PROGRAM BLOCK_CALL
VAR
	CLAMP_1_DB : CLAMP_PROCESS;
	CLAMP_2_DB : CLAMP_PROCESS;
	CLAMP_3_DB : CLAMP_PROCESS;
	CLAMP_4_DB : CLAMP_PROCESS;
	CLAMP_5_DB : CLAMP_PROCESS;
	CLAMP_6_DB : CLAMP_PROCESS;
	Feedback_1_DB : Feedback_FB;
	Feedback_2_DB : Feedback_FB;
	Feedback_3_DB : Feedback_FB;
	Feedback_4_DB : Feedback_FB;
	Feedback_5_DB : Feedback_FB;
	Feedback_6_DB : Feedback_FB;
	Feedback_TT1_DB : Feedback_FB;
	Feedback_Trunion_1_DB : Feedback_FB;
	TURNTABLE_2POS_DB : TURNTABLE_2POS;
	TRUNION1_DB : TRUNION_FB;
	ROLLER_DOOR_DB : ROLLER_DOOR;
	RollerDoor_DB : RollerDoor;
    Feedback_RD1_DB : Feedback_FB;
	WELD_ROBOT_DB : WELD_ROBOT;
	MH_ROBOT_DB : MH_ROBOT;
	MODE_CONTROL_DB : MODE_CONTROL;
	SENSOR_DB : SENSOR;
END_VAR

// note: this text did not pass the execution check against the stored diagram
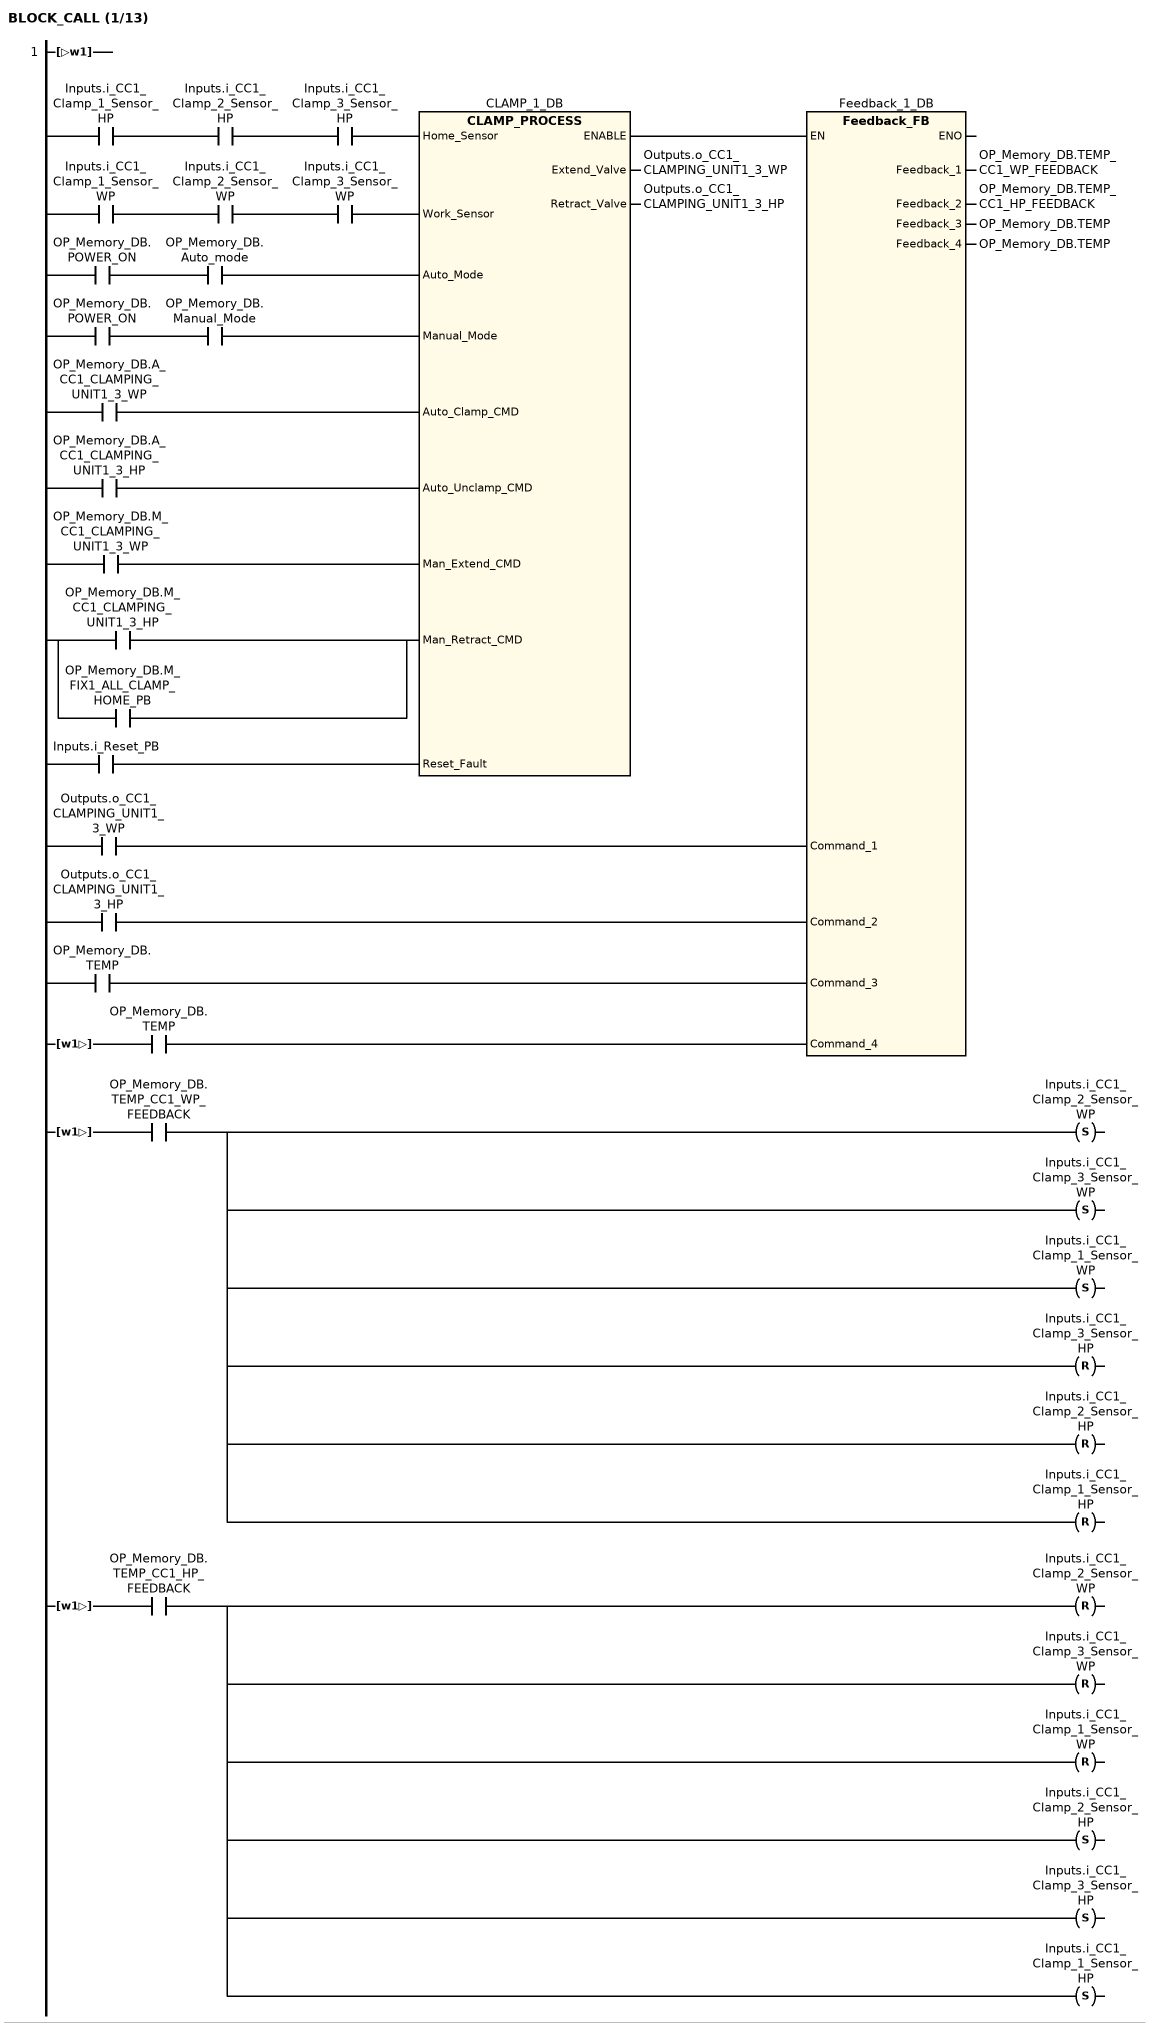
// NETWORK 1
CLAMP_1_DB(
    Home_Sensor := Inputs.i_CC1_Clamp_1_Sensor_HP AND Inputs.i_CC1_Clamp_2_Sensor_HP AND Inputs.i_CC1_Clamp_3_Sensor_HP,
    Work_Sensor := Inputs.i_CC1_Clamp_1_Sensor_WP AND Inputs.i_CC1_Clamp_2_Sensor_WP AND Inputs.i_CC1_Clamp_3_Sensor_WP,
    Auto_Mode := OP_Memory_DB.POWER_ON AND OP_Memory_DB.Auto_mode,
    Manual_Mode := OP_Memory_DB.POWER_ON AND OP_Memory_DB.Manual_Mode,
    Auto_Clamp_CMD := OP_Memory_DB.A_CC1_CLAMPING_UNIT1_3_WP,
    Auto_Unclamp_CMD := OP_Memory_DB.A_CC1_CLAMPING_UNIT1_3_HP,
    Man_Extend_CMD := OP_Memory_DB.M_CC1_CLAMPING_UNIT1_3_WP,
    Man_Retract_CMD := OP_Memory_DB.M_CC1_CLAMPING_UNIT1_3_HP OR OP_Memory_DB.M_FIX1_ALL_CLAMP_HOME_PB,
    Reset_Fault := Inputs.i_Reset_PB,
    Extend_Valve => Outputs.o_CC1_CLAMPING_UNIT1_3_WP,
    Retract_Valve => Outputs.o_CC1_CLAMPING_UNIT1_3_HP); // CLAMP_PROCESS
Feedback_1_DB(
    EN := CLAMP_1_DB.ENABLE,
    Command_1 := Outputs.o_CC1_CLAMPING_UNIT1_3_WP,
    Command_2 := Outputs.o_CC1_CLAMPING_UNIT1_3_HP,
    Command_3 := OP_Memory_DB.TEMP,
    Command_4 := OP_Memory_DB.TEMP,
    Feedback_1 => OP_Memory_DB.TEMP_CC1_WP_FEEDBACK,
    Feedback_2 => OP_Memory_DB.TEMP_CC1_HP_FEEDBACK,
    Feedback_3 => OP_Memory_DB.TEMP,
    Feedback_4 => OP_Memory_DB.TEMP); // Feedback_FB
Inputs.i_CC1_Clamp_2_Sensor_WP S= OP_Memory_DB.TEMP_CC1_WP_FEEDBACK;
Inputs.i_CC1_Clamp_3_Sensor_WP S= OP_Memory_DB.TEMP_CC1_WP_FEEDBACK;
Inputs.i_CC1_Clamp_1_Sensor_WP S= OP_Memory_DB.TEMP_CC1_WP_FEEDBACK;
Inputs.i_CC1_Clamp_3_Sensor_HP R= OP_Memory_DB.TEMP_CC1_WP_FEEDBACK;
Inputs.i_CC1_Clamp_2_Sensor_HP R= OP_Memory_DB.TEMP_CC1_WP_FEEDBACK;
Inputs.i_CC1_Clamp_1_Sensor_HP R= OP_Memory_DB.TEMP_CC1_WP_FEEDBACK;
Inputs.i_CC1_Clamp_2_Sensor_WP R= OP_Memory_DB.TEMP_CC1_HP_FEEDBACK;
Inputs.i_CC1_Clamp_3_Sensor_WP R= OP_Memory_DB.TEMP_CC1_HP_FEEDBACK;
Inputs.i_CC1_Clamp_1_Sensor_WP R= OP_Memory_DB.TEMP_CC1_HP_FEEDBACK;
Inputs.i_CC1_Clamp_2_Sensor_HP S= OP_Memory_DB.TEMP_CC1_HP_FEEDBACK;
Inputs.i_CC1_Clamp_3_Sensor_HP S= OP_Memory_DB.TEMP_CC1_HP_FEEDBACK;
Inputs.i_CC1_Clamp_1_Sensor_HP S= OP_Memory_DB.TEMP_CC1_HP_FEEDBACK;

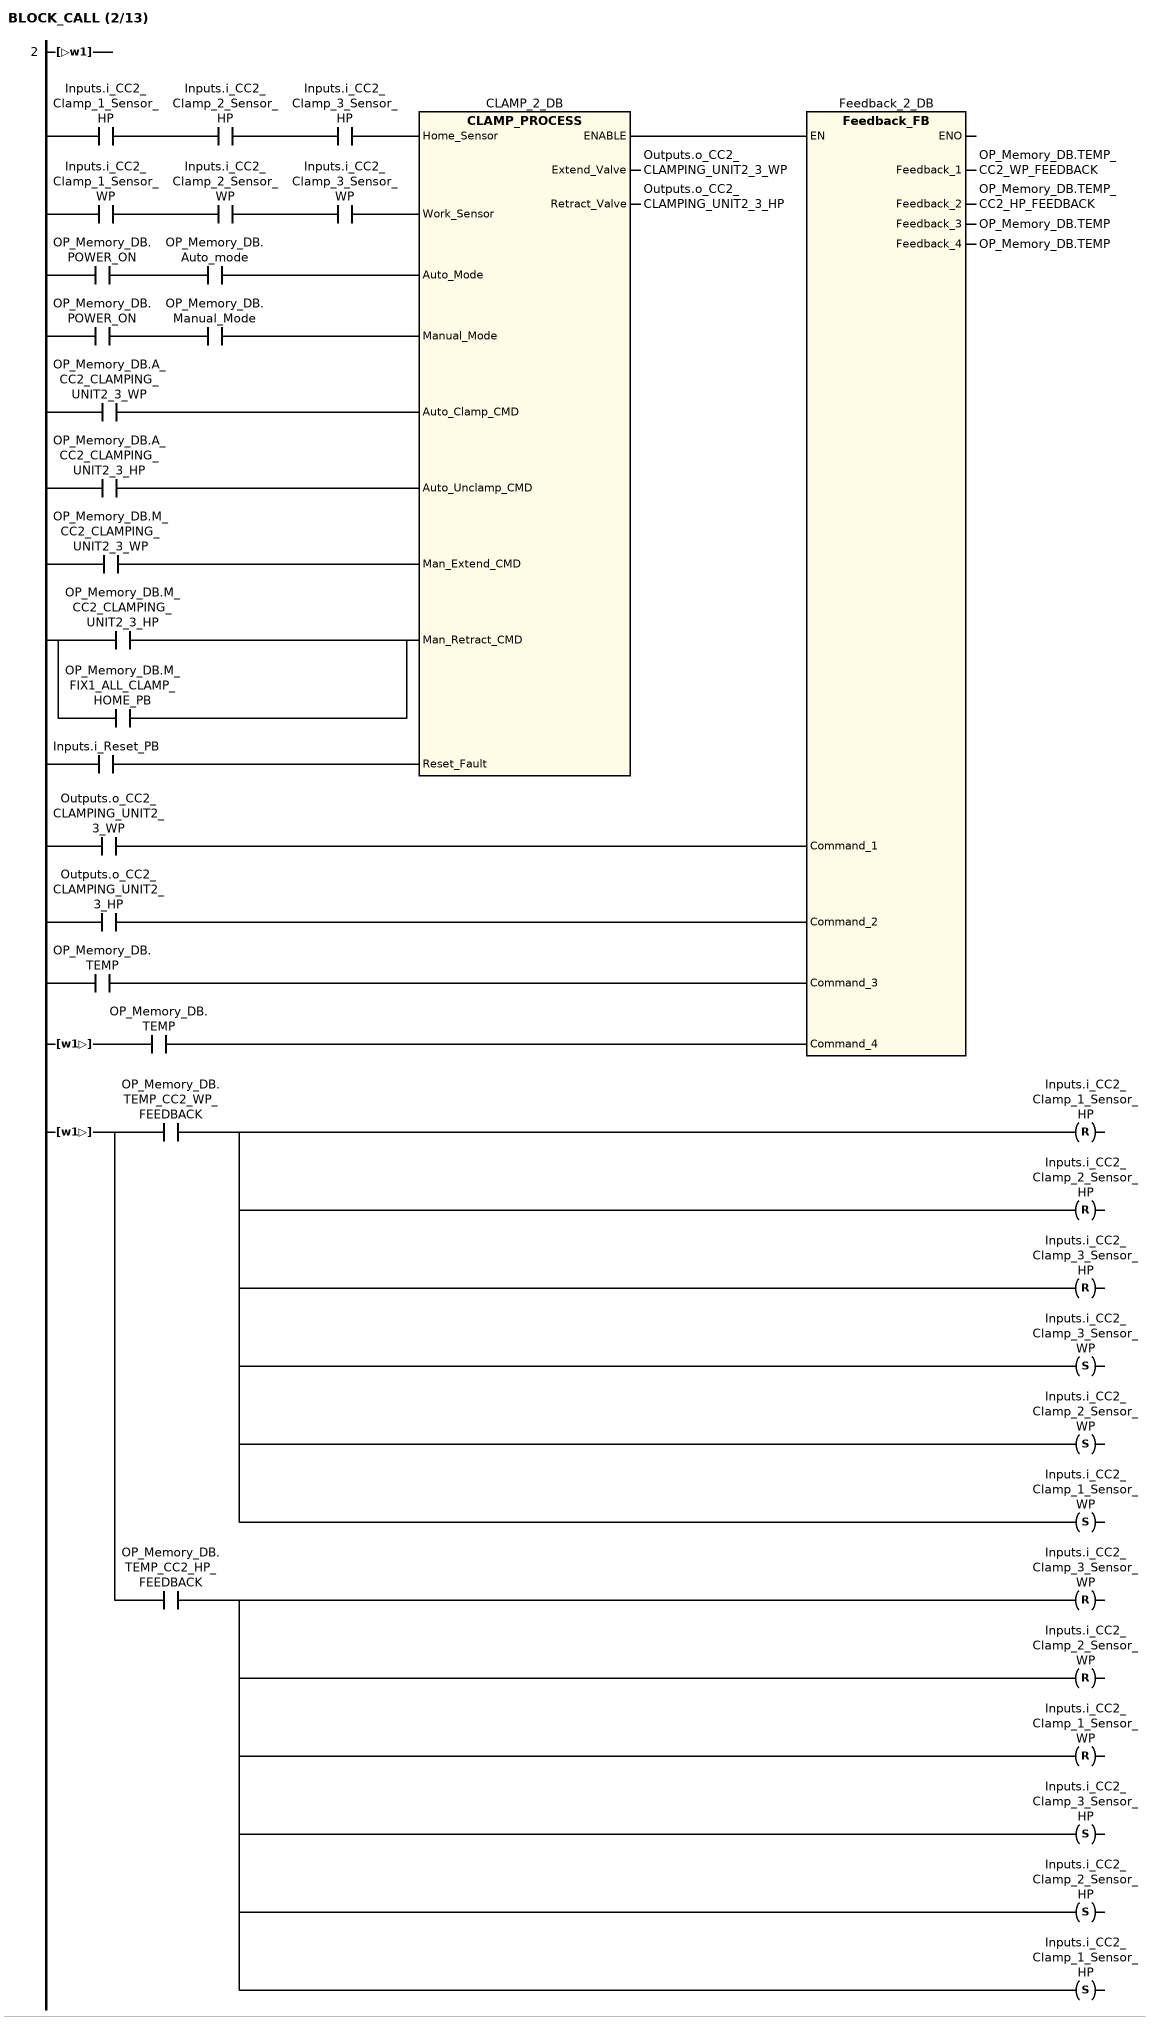
// NETWORK 2
CLAMP_2_DB(
    Home_Sensor := Inputs.i_CC2_Clamp_1_Sensor_HP AND Inputs.i_CC2_Clamp_2_Sensor_HP AND Inputs.i_CC2_Clamp_3_Sensor_HP,
    Work_Sensor := Inputs.i_CC2_Clamp_1_Sensor_WP AND Inputs.i_CC2_Clamp_2_Sensor_WP AND Inputs.i_CC2_Clamp_3_Sensor_WP,
    Auto_Mode := OP_Memory_DB.POWER_ON AND OP_Memory_DB.Auto_mode,
    Manual_Mode := OP_Memory_DB.POWER_ON AND OP_Memory_DB.Manual_Mode,
    Auto_Clamp_CMD := OP_Memory_DB.A_CC2_CLAMPING_UNIT2_3_WP,
    Auto_Unclamp_CMD := OP_Memory_DB.A_CC2_CLAMPING_UNIT2_3_HP,
    Man_Extend_CMD := OP_Memory_DB.M_CC2_CLAMPING_UNIT2_3_WP,
    Man_Retract_CMD := OP_Memory_DB.M_CC2_CLAMPING_UNIT2_3_HP OR OP_Memory_DB.M_FIX1_ALL_CLAMP_HOME_PB,
    Reset_Fault := Inputs.i_Reset_PB,
    Extend_Valve => Outputs.o_CC2_CLAMPING_UNIT2_3_WP,
    Retract_Valve => Outputs.o_CC2_CLAMPING_UNIT2_3_HP); // CLAMP_PROCESS
Feedback_2_DB(
    EN := CLAMP_2_DB.ENABLE,
    Command_1 := Outputs.o_CC2_CLAMPING_UNIT2_3_WP,
    Command_2 := Outputs.o_CC2_CLAMPING_UNIT2_3_HP,
    Command_3 := OP_Memory_DB.TEMP,
    Command_4 := OP_Memory_DB.TEMP,
    Feedback_1 => OP_Memory_DB.TEMP_CC2_WP_FEEDBACK,
    Feedback_2 => OP_Memory_DB.TEMP_CC2_HP_FEEDBACK,
    Feedback_3 => OP_Memory_DB.TEMP,
    Feedback_4 => OP_Memory_DB.TEMP); // Feedback_FB
Inputs.i_CC2_Clamp_1_Sensor_HP R= OP_Memory_DB.TEMP_CC2_WP_FEEDBACK;
Inputs.i_CC2_Clamp_2_Sensor_HP R= OP_Memory_DB.TEMP_CC2_WP_FEEDBACK;
Inputs.i_CC2_Clamp_3_Sensor_HP R= OP_Memory_DB.TEMP_CC2_WP_FEEDBACK;
Inputs.i_CC2_Clamp_3_Sensor_WP S= OP_Memory_DB.TEMP_CC2_WP_FEEDBACK;
Inputs.i_CC2_Clamp_2_Sensor_WP S= OP_Memory_DB.TEMP_CC2_WP_FEEDBACK;
Inputs.i_CC2_Clamp_1_Sensor_WP S= OP_Memory_DB.TEMP_CC2_WP_FEEDBACK;
Inputs.i_CC2_Clamp_3_Sensor_WP R= OP_Memory_DB.TEMP_CC2_HP_FEEDBACK;
Inputs.i_CC2_Clamp_2_Sensor_WP R= OP_Memory_DB.TEMP_CC2_HP_FEEDBACK;
Inputs.i_CC2_Clamp_1_Sensor_WP R= OP_Memory_DB.TEMP_CC2_HP_FEEDBACK;
Inputs.i_CC2_Clamp_3_Sensor_HP S= OP_Memory_DB.TEMP_CC2_HP_FEEDBACK;
Inputs.i_CC2_Clamp_2_Sensor_HP S= OP_Memory_DB.TEMP_CC2_HP_FEEDBACK;
Inputs.i_CC2_Clamp_1_Sensor_HP S= OP_Memory_DB.TEMP_CC2_HP_FEEDBACK;

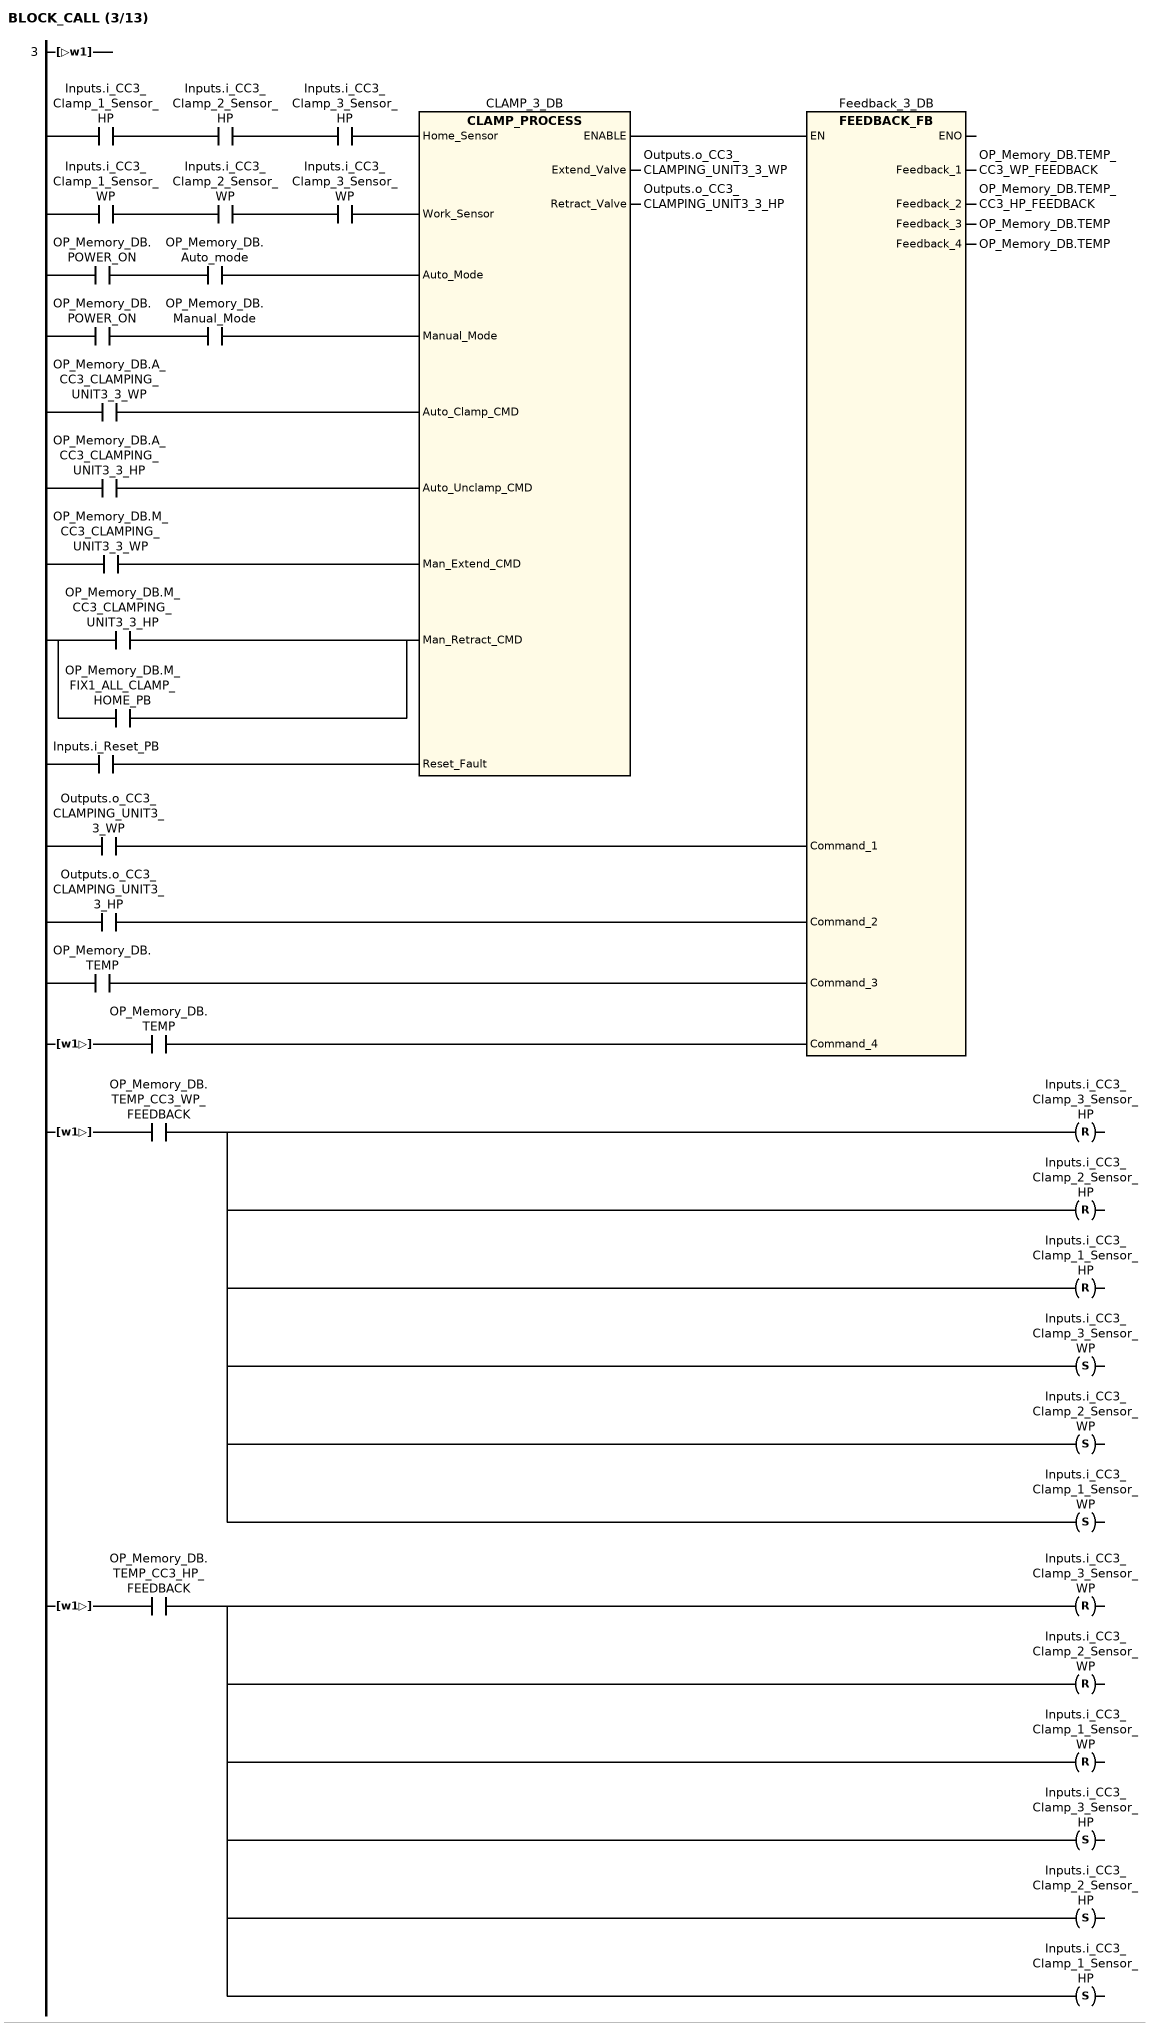
// NETWORK 3
CLAMP_3_DB(
    Home_Sensor := Inputs.i_CC3_Clamp_1_Sensor_HP AND Inputs.i_CC3_Clamp_2_Sensor_HP AND Inputs.i_CC3_Clamp_3_Sensor_HP,
    Work_Sensor := Inputs.i_CC3_Clamp_1_Sensor_WP AND Inputs.i_CC3_Clamp_2_Sensor_WP AND Inputs.i_CC3_Clamp_3_Sensor_WP,
    Auto_Mode := OP_Memory_DB.POWER_ON AND OP_Memory_DB.Auto_mode,
    Manual_Mode := OP_Memory_DB.POWER_ON AND OP_Memory_DB.Manual_Mode,
    Auto_Clamp_CMD := OP_Memory_DB.A_CC3_CLAMPING_UNIT3_3_WP,
    Auto_Unclamp_CMD := OP_Memory_DB.A_CC3_CLAMPING_UNIT3_3_HP,
    Man_Extend_CMD := OP_Memory_DB.M_CC3_CLAMPING_UNIT3_3_WP,
    Man_Retract_CMD := OP_Memory_DB.M_CC3_CLAMPING_UNIT3_3_HP OR OP_Memory_DB.M_FIX1_ALL_CLAMP_HOME_PB,
    Reset_Fault := Inputs.i_Reset_PB,
    Extend_Valve => Outputs.o_CC3_CLAMPING_UNIT3_3_WP,
    Retract_Valve => Outputs.o_CC3_CLAMPING_UNIT3_3_HP); // CLAMP_PROCESS
Feedback_3_DB(
    EN := CLAMP_3_DB.ENABLE,
    Command_1 := Outputs.o_CC3_CLAMPING_UNIT3_3_WP,
    Command_2 := Outputs.o_CC3_CLAMPING_UNIT3_3_HP,
    Command_3 := OP_Memory_DB.TEMP,
    Command_4 := OP_Memory_DB.TEMP,
    Feedback_1 => OP_Memory_DB.TEMP_CC3_WP_FEEDBACK,
    Feedback_2 => OP_Memory_DB.TEMP_CC3_HP_FEEDBACK,
    Feedback_3 => OP_Memory_DB.TEMP,
    Feedback_4 => OP_Memory_DB.TEMP); // FEEDBACK_FB
Inputs.i_CC3_Clamp_3_Sensor_HP R= OP_Memory_DB.TEMP_CC3_WP_FEEDBACK;
Inputs.i_CC3_Clamp_2_Sensor_HP R= OP_Memory_DB.TEMP_CC3_WP_FEEDBACK;
Inputs.i_CC3_Clamp_1_Sensor_HP R= OP_Memory_DB.TEMP_CC3_WP_FEEDBACK;
Inputs.i_CC3_Clamp_3_Sensor_WP S= OP_Memory_DB.TEMP_CC3_WP_FEEDBACK;
Inputs.i_CC3_Clamp_2_Sensor_WP S= OP_Memory_DB.TEMP_CC3_WP_FEEDBACK;
Inputs.i_CC3_Clamp_1_Sensor_WP S= OP_Memory_DB.TEMP_CC3_WP_FEEDBACK;
Inputs.i_CC3_Clamp_3_Sensor_WP R= OP_Memory_DB.TEMP_CC3_HP_FEEDBACK;
Inputs.i_CC3_Clamp_2_Sensor_WP R= OP_Memory_DB.TEMP_CC3_HP_FEEDBACK;
Inputs.i_CC3_Clamp_1_Sensor_WP R= OP_Memory_DB.TEMP_CC3_HP_FEEDBACK;
Inputs.i_CC3_Clamp_3_Sensor_HP S= OP_Memory_DB.TEMP_CC3_HP_FEEDBACK;
Inputs.i_CC3_Clamp_2_Sensor_HP S= OP_Memory_DB.TEMP_CC3_HP_FEEDBACK;
Inputs.i_CC3_Clamp_1_Sensor_HP S= OP_Memory_DB.TEMP_CC3_HP_FEEDBACK;

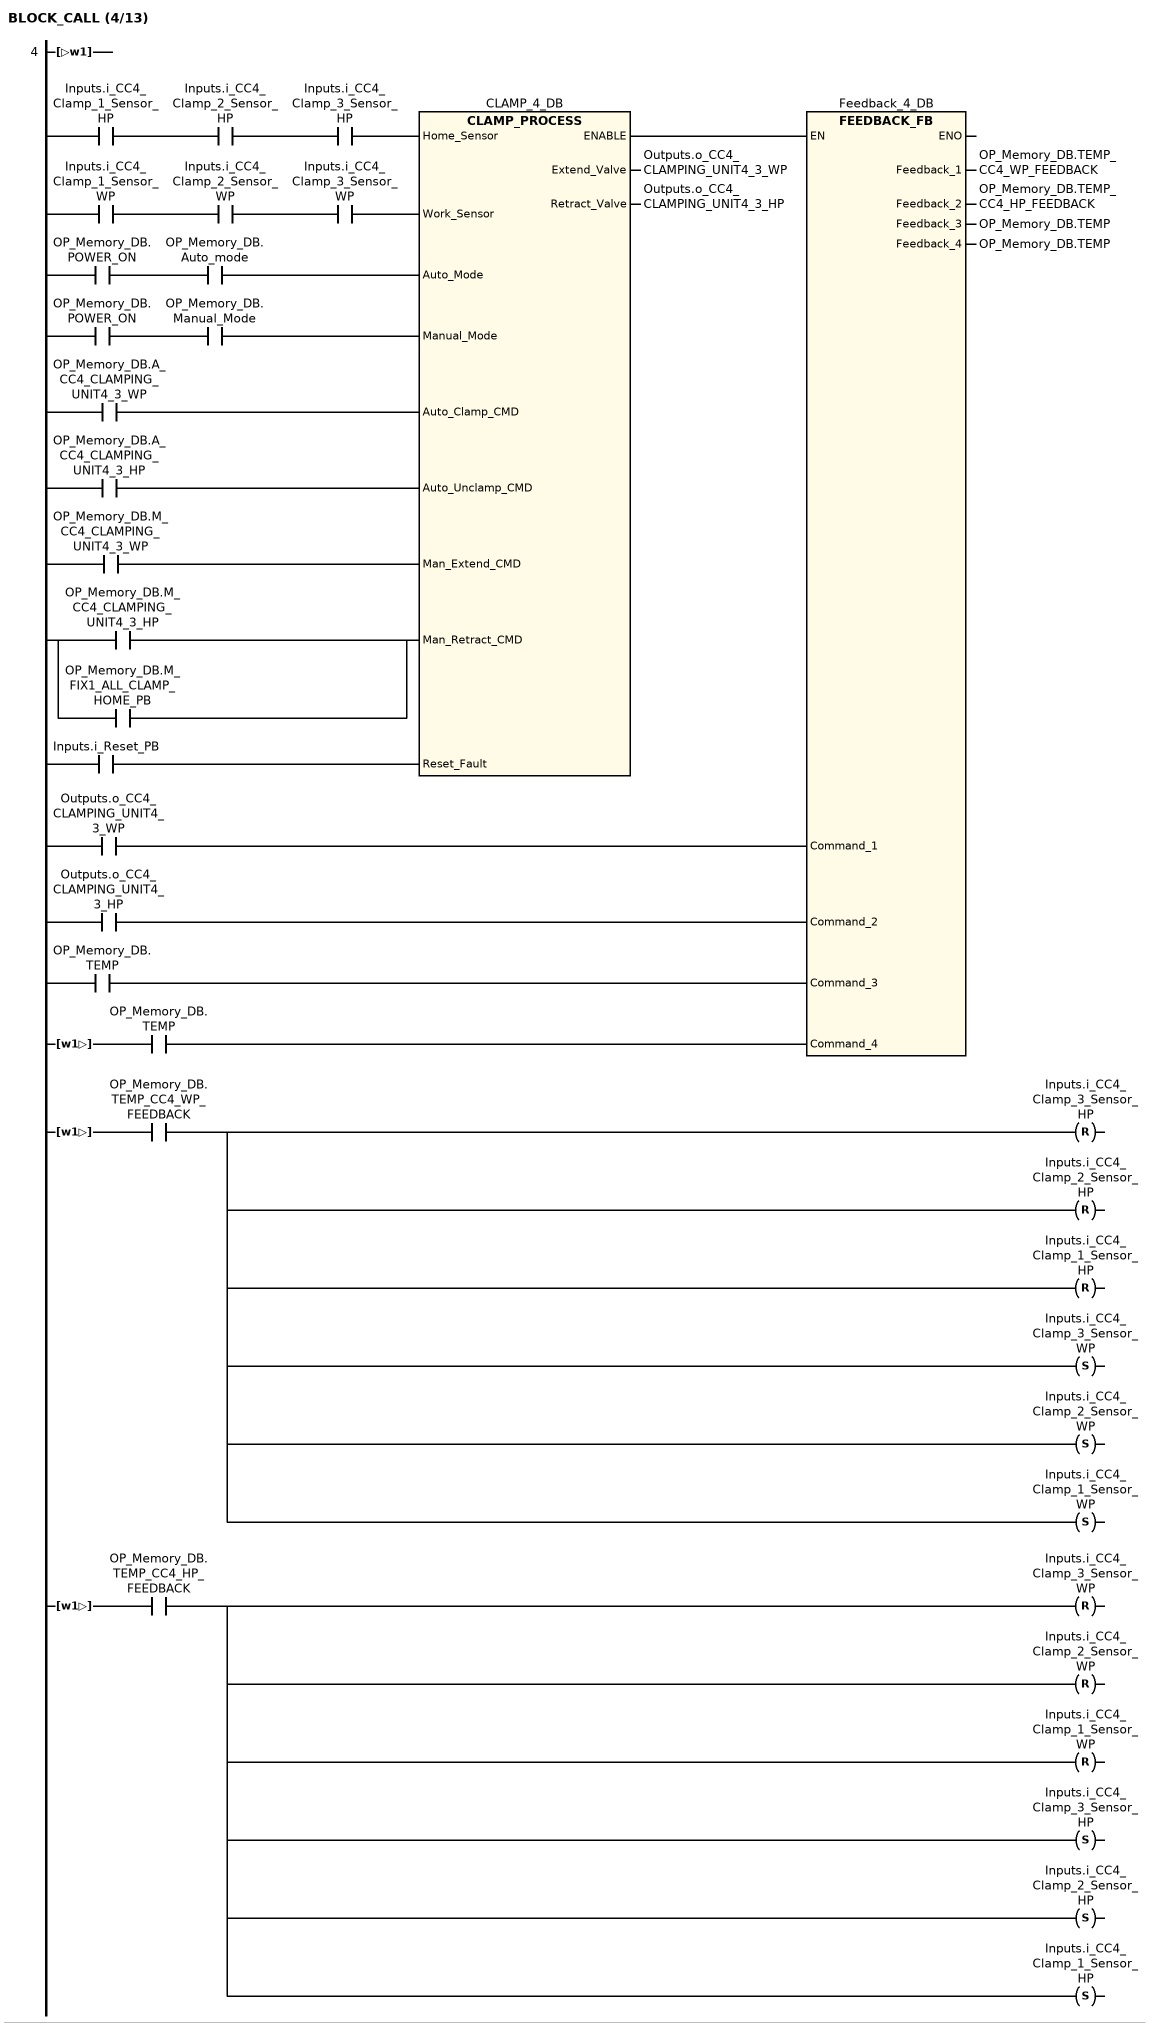
// NETWORK 4
CLAMP_4_DB(
    Home_Sensor := Inputs.i_CC4_Clamp_1_Sensor_HP AND Inputs.i_CC4_Clamp_2_Sensor_HP AND Inputs.i_CC4_Clamp_3_Sensor_HP,
    Work_Sensor := Inputs.i_CC4_Clamp_1_Sensor_WP AND Inputs.i_CC4_Clamp_2_Sensor_WP AND Inputs.i_CC4_Clamp_3_Sensor_WP,
    Auto_Mode := OP_Memory_DB.POWER_ON AND OP_Memory_DB.Auto_mode,
    Manual_Mode := OP_Memory_DB.POWER_ON AND OP_Memory_DB.Manual_Mode,
    Auto_Clamp_CMD := OP_Memory_DB.A_CC4_CLAMPING_UNIT4_3_WP,
    Auto_Unclamp_CMD := OP_Memory_DB.A_CC4_CLAMPING_UNIT4_3_HP,
    Man_Extend_CMD := OP_Memory_DB.M_CC4_CLAMPING_UNIT4_3_WP,
    Man_Retract_CMD := OP_Memory_DB.M_CC4_CLAMPING_UNIT4_3_HP OR OP_Memory_DB.M_FIX1_ALL_CLAMP_HOME_PB,
    Reset_Fault := Inputs.i_Reset_PB,
    Extend_Valve => Outputs.o_CC4_CLAMPING_UNIT4_3_WP,
    Retract_Valve => Outputs.o_CC4_CLAMPING_UNIT4_3_HP); // CLAMP_PROCESS
Feedback_4_DB(
    EN := CLAMP_4_DB.ENABLE,
    Command_1 := Outputs.o_CC4_CLAMPING_UNIT4_3_WP,
    Command_2 := Outputs.o_CC4_CLAMPING_UNIT4_3_HP,
    Command_3 := OP_Memory_DB.TEMP,
    Command_4 := OP_Memory_DB.TEMP,
    Feedback_1 => OP_Memory_DB.TEMP_CC4_WP_FEEDBACK,
    Feedback_2 => OP_Memory_DB.TEMP_CC4_HP_FEEDBACK,
    Feedback_3 => OP_Memory_DB.TEMP,
    Feedback_4 => OP_Memory_DB.TEMP); // FEEDBACK_FB
Inputs.i_CC4_Clamp_3_Sensor_HP R= OP_Memory_DB.TEMP_CC4_WP_FEEDBACK;
Inputs.i_CC4_Clamp_2_Sensor_HP R= OP_Memory_DB.TEMP_CC4_WP_FEEDBACK;
Inputs.i_CC4_Clamp_1_Sensor_HP R= OP_Memory_DB.TEMP_CC4_WP_FEEDBACK;
Inputs.i_CC4_Clamp_3_Sensor_WP S= OP_Memory_DB.TEMP_CC4_WP_FEEDBACK;
Inputs.i_CC4_Clamp_2_Sensor_WP S= OP_Memory_DB.TEMP_CC4_WP_FEEDBACK;
Inputs.i_CC4_Clamp_1_Sensor_WP S= OP_Memory_DB.TEMP_CC4_WP_FEEDBACK;
Inputs.i_CC4_Clamp_3_Sensor_WP R= OP_Memory_DB.TEMP_CC4_HP_FEEDBACK;
Inputs.i_CC4_Clamp_2_Sensor_WP R= OP_Memory_DB.TEMP_CC4_HP_FEEDBACK;
Inputs.i_CC4_Clamp_1_Sensor_WP R= OP_Memory_DB.TEMP_CC4_HP_FEEDBACK;
Inputs.i_CC4_Clamp_3_Sensor_HP S= OP_Memory_DB.TEMP_CC4_HP_FEEDBACK;
Inputs.i_CC4_Clamp_2_Sensor_HP S= OP_Memory_DB.TEMP_CC4_HP_FEEDBACK;
Inputs.i_CC4_Clamp_1_Sensor_HP S= OP_Memory_DB.TEMP_CC4_HP_FEEDBACK;

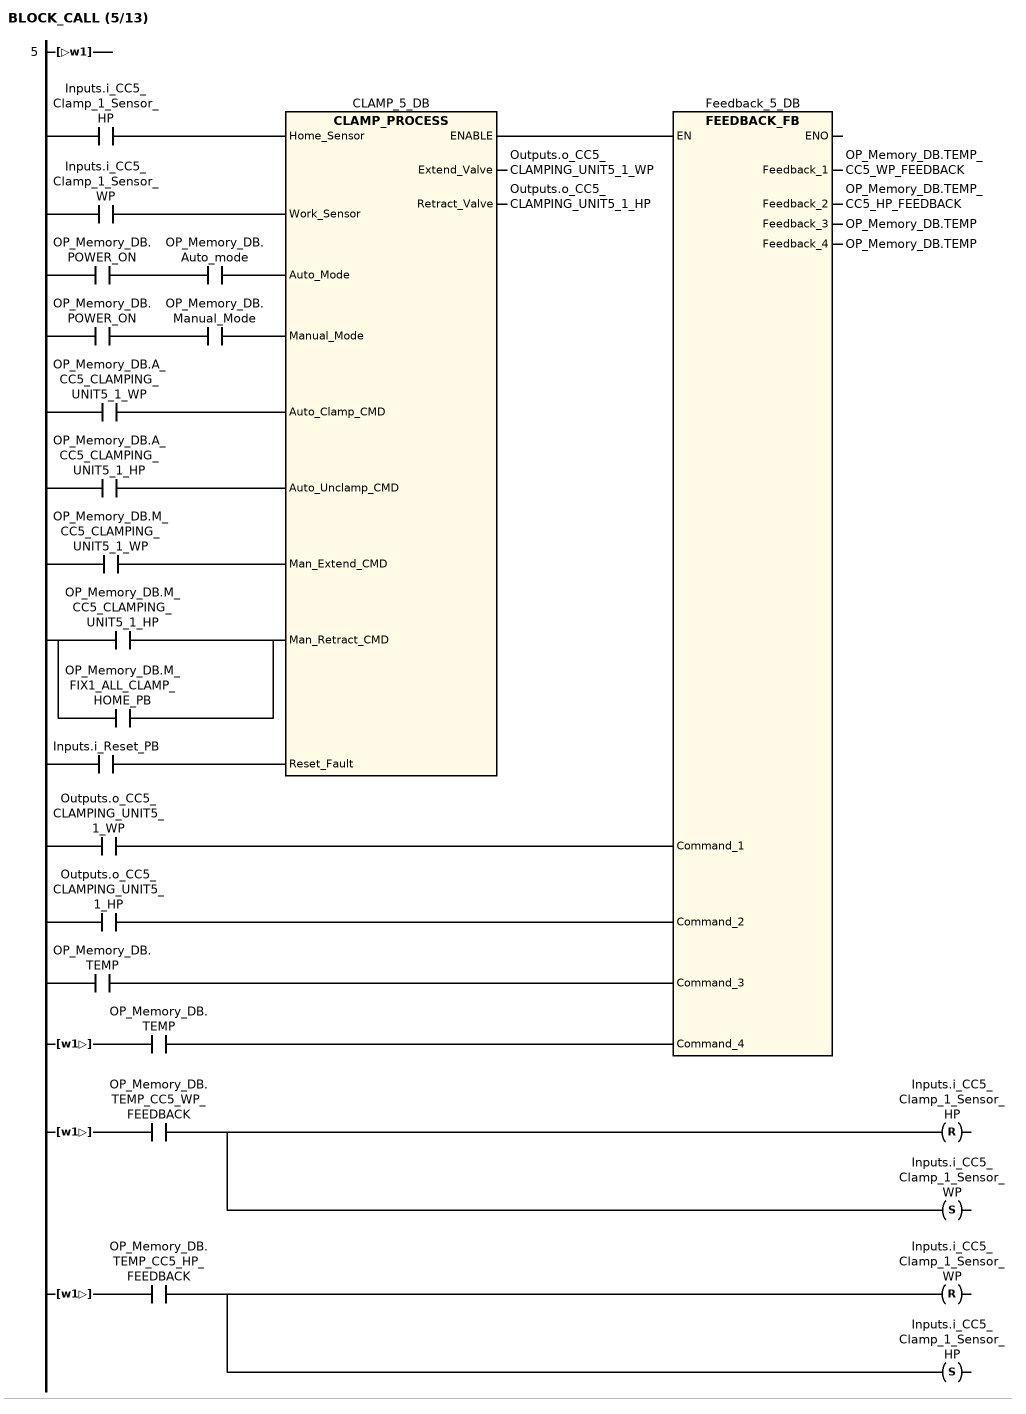
// NETWORK 5
CLAMP_5_DB(
    Home_Sensor := Inputs.i_CC5_Clamp_1_Sensor_HP,
    Work_Sensor := Inputs.i_CC5_Clamp_1_Sensor_WP,
    Auto_Mode := OP_Memory_DB.POWER_ON AND OP_Memory_DB.Auto_mode,
    Manual_Mode := OP_Memory_DB.POWER_ON AND OP_Memory_DB.Manual_Mode,
    Auto_Clamp_CMD := OP_Memory_DB.A_CC5_CLAMPING_UNIT5_1_WP,
    Auto_Unclamp_CMD := OP_Memory_DB.A_CC5_CLAMPING_UNIT5_1_HP,
    Man_Extend_CMD := OP_Memory_DB.M_CC5_CLAMPING_UNIT5_1_WP,
    Man_Retract_CMD := OP_Memory_DB.M_CC5_CLAMPING_UNIT5_1_HP OR OP_Memory_DB.M_FIX1_ALL_CLAMP_HOME_PB,
    Reset_Fault := Inputs.i_Reset_PB,
    Extend_Valve => Outputs.o_CC5_CLAMPING_UNIT5_1_WP,
    Retract_Valve => Outputs.o_CC5_CLAMPING_UNIT5_1_HP); // CLAMP_PROCESS
Feedback_5_DB(
    EN := CLAMP_5_DB.ENABLE,
    Command_1 := Outputs.o_CC5_CLAMPING_UNIT5_1_WP,
    Command_2 := Outputs.o_CC5_CLAMPING_UNIT5_1_HP,
    Command_3 := OP_Memory_DB.TEMP,
    Command_4 := OP_Memory_DB.TEMP,
    Feedback_1 => OP_Memory_DB.TEMP_CC5_WP_FEEDBACK,
    Feedback_2 => OP_Memory_DB.TEMP_CC5_HP_FEEDBACK,
    Feedback_3 => OP_Memory_DB.TEMP,
    Feedback_4 => OP_Memory_DB.TEMP); // FEEDBACK_FB
Inputs.i_CC5_Clamp_1_Sensor_HP R= OP_Memory_DB.TEMP_CC5_WP_FEEDBACK;
Inputs.i_CC5_Clamp_1_Sensor_WP S= OP_Memory_DB.TEMP_CC5_WP_FEEDBACK;
Inputs.i_CC5_Clamp_1_Sensor_WP R= OP_Memory_DB.TEMP_CC5_HP_FEEDBACK;
Inputs.i_CC5_Clamp_1_Sensor_HP S= OP_Memory_DB.TEMP_CC5_HP_FEEDBACK;

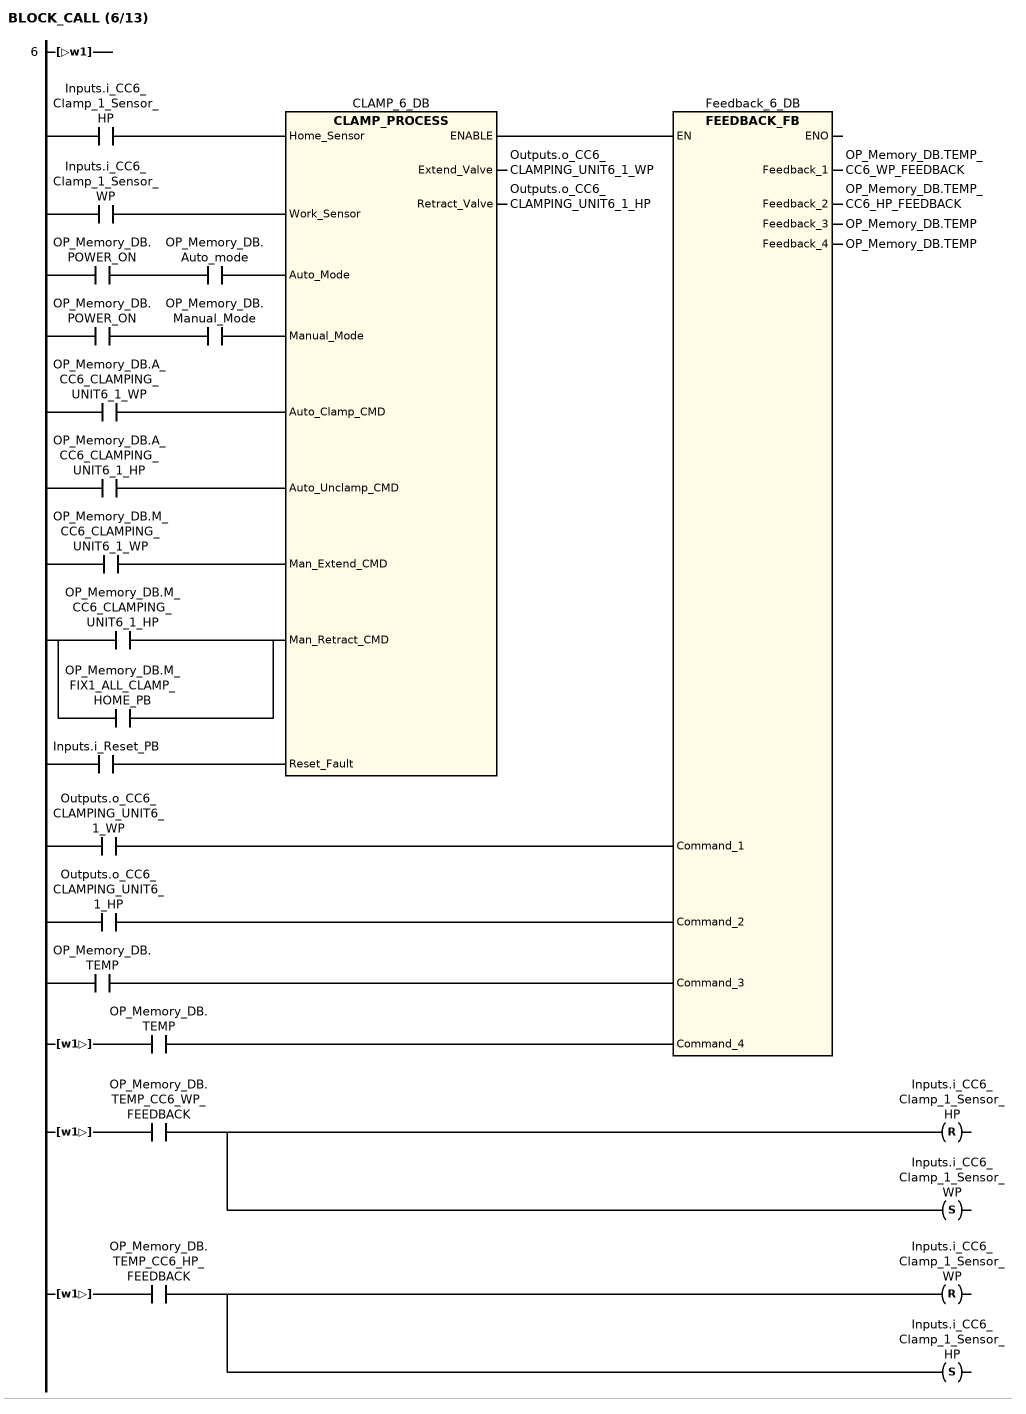
// NETWORK 6
CLAMP_6_DB(
    Home_Sensor := Inputs.i_CC6_Clamp_1_Sensor_HP,
    Work_Sensor := Inputs.i_CC6_Clamp_1_Sensor_WP,
    Auto_Mode := OP_Memory_DB.POWER_ON AND OP_Memory_DB.Auto_mode,
    Manual_Mode := OP_Memory_DB.POWER_ON AND OP_Memory_DB.Manual_Mode,
    Auto_Clamp_CMD := OP_Memory_DB.A_CC6_CLAMPING_UNIT6_1_WP,
    Auto_Unclamp_CMD := OP_Memory_DB.A_CC6_CLAMPING_UNIT6_1_HP,
    Man_Extend_CMD := OP_Memory_DB.M_CC6_CLAMPING_UNIT6_1_WP,
    Man_Retract_CMD := OP_Memory_DB.M_CC6_CLAMPING_UNIT6_1_HP OR OP_Memory_DB.M_FIX1_ALL_CLAMP_HOME_PB,
    Reset_Fault := Inputs.i_Reset_PB,
    Extend_Valve => Outputs.o_CC6_CLAMPING_UNIT6_1_WP,
    Retract_Valve => Outputs.o_CC6_CLAMPING_UNIT6_1_HP); // CLAMP_PROCESS
Feedback_6_DB(
    EN := CLAMP_6_DB.ENABLE,
    Command_1 := Outputs.o_CC6_CLAMPING_UNIT6_1_WP,
    Command_2 := Outputs.o_CC6_CLAMPING_UNIT6_1_HP,
    Command_3 := OP_Memory_DB.TEMP,
    Command_4 := OP_Memory_DB.TEMP,
    Feedback_1 => OP_Memory_DB.TEMP_CC6_WP_FEEDBACK,
    Feedback_2 => OP_Memory_DB.TEMP_CC6_HP_FEEDBACK,
    Feedback_3 => OP_Memory_DB.TEMP,
    Feedback_4 => OP_Memory_DB.TEMP); // FEEDBACK_FB
Inputs.i_CC6_Clamp_1_Sensor_HP R= OP_Memory_DB.TEMP_CC6_WP_FEEDBACK;
Inputs.i_CC6_Clamp_1_Sensor_WP S= OP_Memory_DB.TEMP_CC6_WP_FEEDBACK;
Inputs.i_CC6_Clamp_1_Sensor_WP R= OP_Memory_DB.TEMP_CC6_HP_FEEDBACK;
Inputs.i_CC6_Clamp_1_Sensor_HP S= OP_Memory_DB.TEMP_CC6_HP_FEEDBACK;

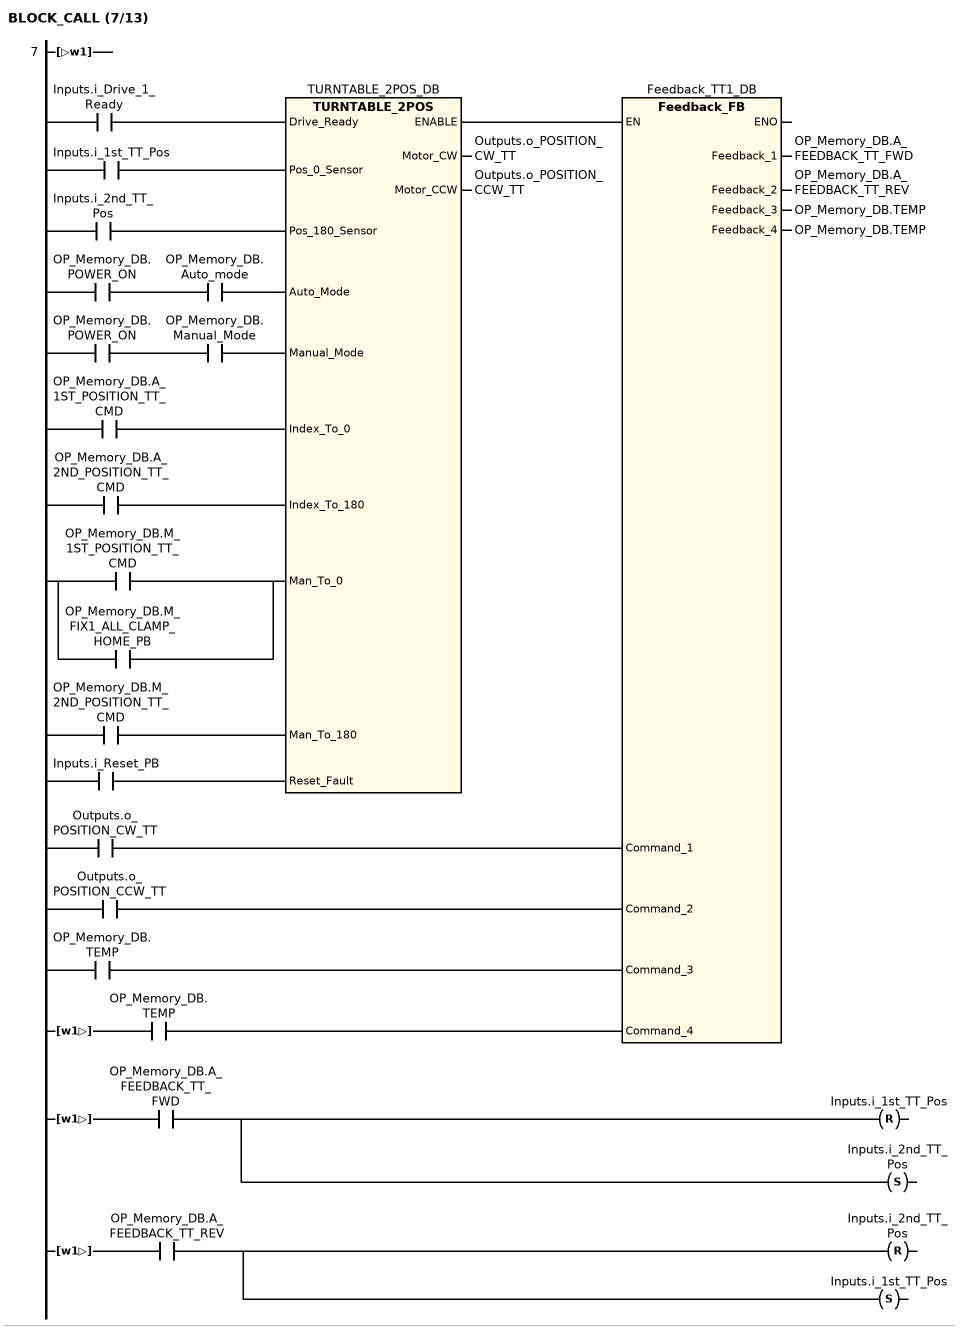
// NETWORK 7
TURNTABLE_2POS_DB(
    Drive_Ready := Inputs.i_Drive_1_Ready,
    Pos_0_Sensor := Inputs.i_1st_TT_Pos,
    Pos_180_Sensor := Inputs.i_2nd_TT_Pos,
    Auto_Mode := OP_Memory_DB.POWER_ON AND OP_Memory_DB.Auto_mode,
    Manual_Mode := OP_Memory_DB.POWER_ON AND OP_Memory_DB.Manual_Mode,
    Index_To_0 := OP_Memory_DB.A_1ST_POSITION_TT_CMD,
    Index_To_180 := OP_Memory_DB.A_2ND_POSITION_TT_CMD,
    Man_To_0 := OP_Memory_DB.M_1ST_POSITION_TT_CMD OR OP_Memory_DB.M_FIX1_ALL_CLAMP_HOME_PB,
    Man_To_180 := OP_Memory_DB.M_2ND_POSITION_TT_CMD,
    Reset_Fault := Inputs.i_Reset_PB,
    Motor_CW => Outputs.o_POSITION_CW_TT,
    Motor_CCW => Outputs.o_POSITION_CCW_TT); // TURNTABLE_2POS
Feedback_TT1_DB(
    EN := TURNTABLE_2POS_DB.ENABLE,
    Command_1 := Outputs.o_POSITION_CW_TT,
    Command_2 := Outputs.o_POSITION_CCW_TT,
    Command_3 := OP_Memory_DB.TEMP,
    Command_4 := OP_Memory_DB.TEMP,
    Feedback_1 => OP_Memory_DB.A_FEEDBACK_TT_FWD,
    Feedback_2 => OP_Memory_DB.A_FEEDBACK_TT_REV,
    Feedback_3 => OP_Memory_DB.TEMP,
    Feedback_4 => OP_Memory_DB.TEMP); // Feedback_FB
Inputs.i_1st_TT_Pos R= OP_Memory_DB.A_FEEDBACK_TT_FWD;
Inputs.i_2nd_TT_Pos S= OP_Memory_DB.A_FEEDBACK_TT_FWD;
Inputs.i_2nd_TT_Pos R= OP_Memory_DB.A_FEEDBACK_TT_REV;
Inputs.i_1st_TT_Pos S= OP_Memory_DB.A_FEEDBACK_TT_REV;

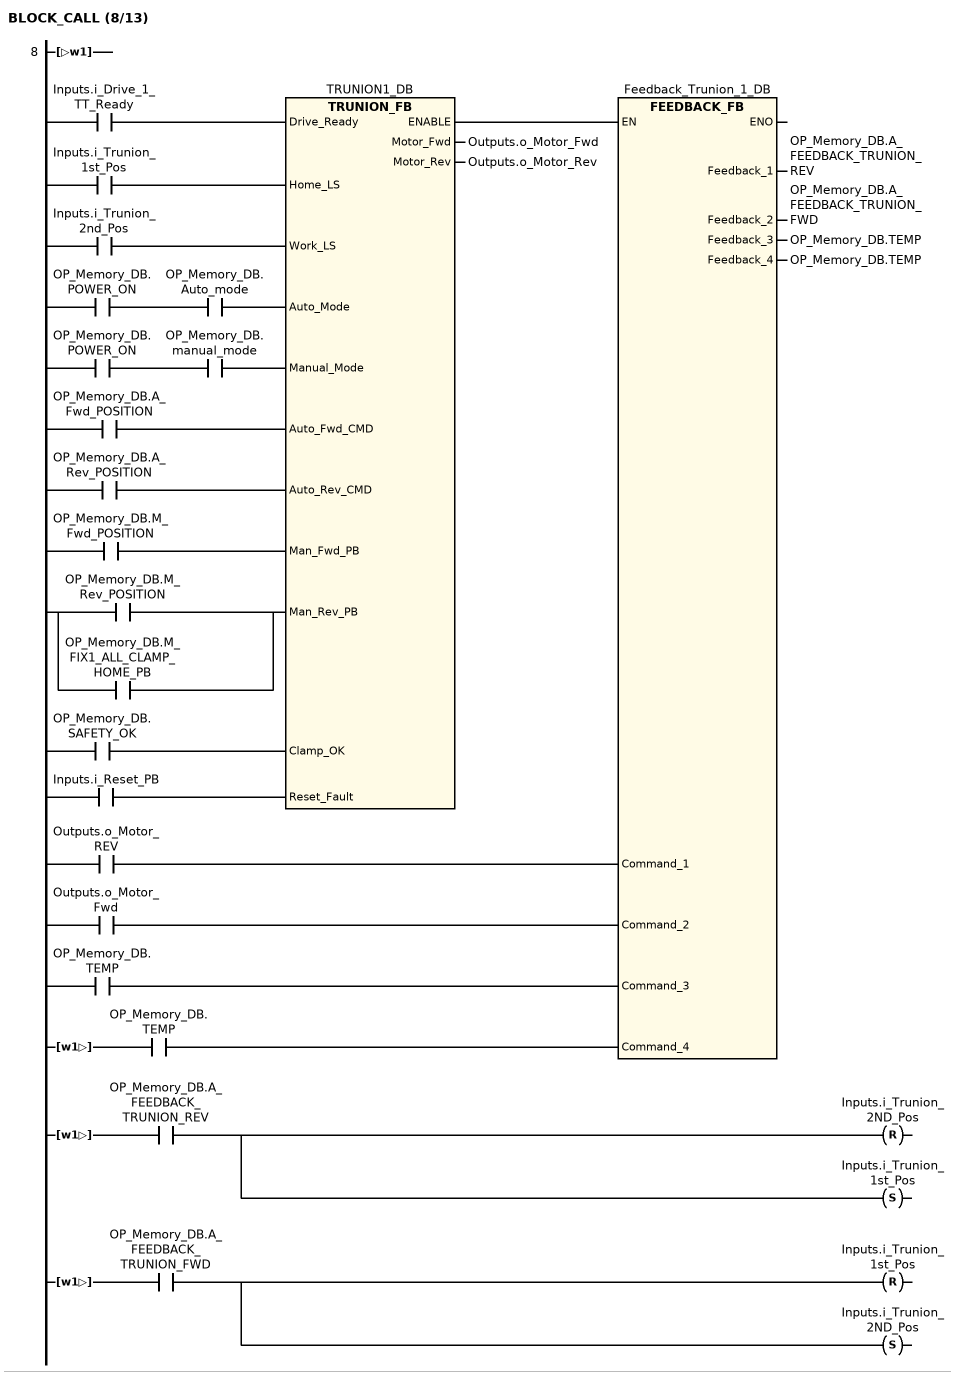
// NETWORK 8
TRUNION1_DB(
    Drive_Ready := Inputs.i_Drive_1_TT_Ready,
    Home_LS := Inputs.i_Trunion_1st_Pos,
    Work_LS := Inputs.i_Trunion_2nd_Pos,
    Auto_Mode := OP_Memory_DB.POWER_ON AND OP_Memory_DB.Auto_mode,
    Manual_Mode := OP_Memory_DB.POWER_ON AND OP_Memory_DB.manual_mode,
    Auto_Fwd_CMD := OP_Memory_DB.A_Fwd_POSITION,
    Auto_Rev_CMD := OP_Memory_DB.A_Rev_POSITION,
    Man_Fwd_PB := OP_Memory_DB.M_Fwd_POSITION,
    Man_Rev_PB := OP_Memory_DB.M_Rev_POSITION OR OP_Memory_DB.M_FIX1_ALL_CLAMP_HOME_PB,
    Clamp_OK := OP_Memory_DB.SAFETY_OK,
    Reset_Fault := Inputs.i_Reset_PB,
    Motor_Fwd => Outputs.o_Motor_Fwd,
    Motor_Rev => Outputs.o_Motor_Rev); // TRUNION_FB
Feedback_Trunion_1_DB(
    EN := TRUNION1_DB.ENABLE,
    Command_1 := Outputs.o_Motor_REV,
    Command_2 := Outputs.o_Motor_Fwd,
    Command_3 := OP_Memory_DB.TEMP,
    Command_4 := OP_Memory_DB.TEMP,
    Feedback_1 => OP_Memory_DB.A_FEEDBACK_TRUNION_REV,
    Feedback_2 => OP_Memory_DB.A_FEEDBACK_TRUNION_FWD,
    Feedback_3 => OP_Memory_DB.TEMP,
    Feedback_4 => OP_Memory_DB.TEMP); // FEEDBACK_FB
Inputs.i_Trunion_2ND_Pos R= OP_Memory_DB.A_FEEDBACK_TRUNION_REV;
Inputs.i_Trunion_1st_Pos S= OP_Memory_DB.A_FEEDBACK_TRUNION_REV;
Inputs.i_Trunion_1st_Pos R= OP_Memory_DB.A_FEEDBACK_TRUNION_FWD;
Inputs.i_Trunion_2ND_Pos S= OP_Memory_DB.A_FEEDBACK_TRUNION_FWD;

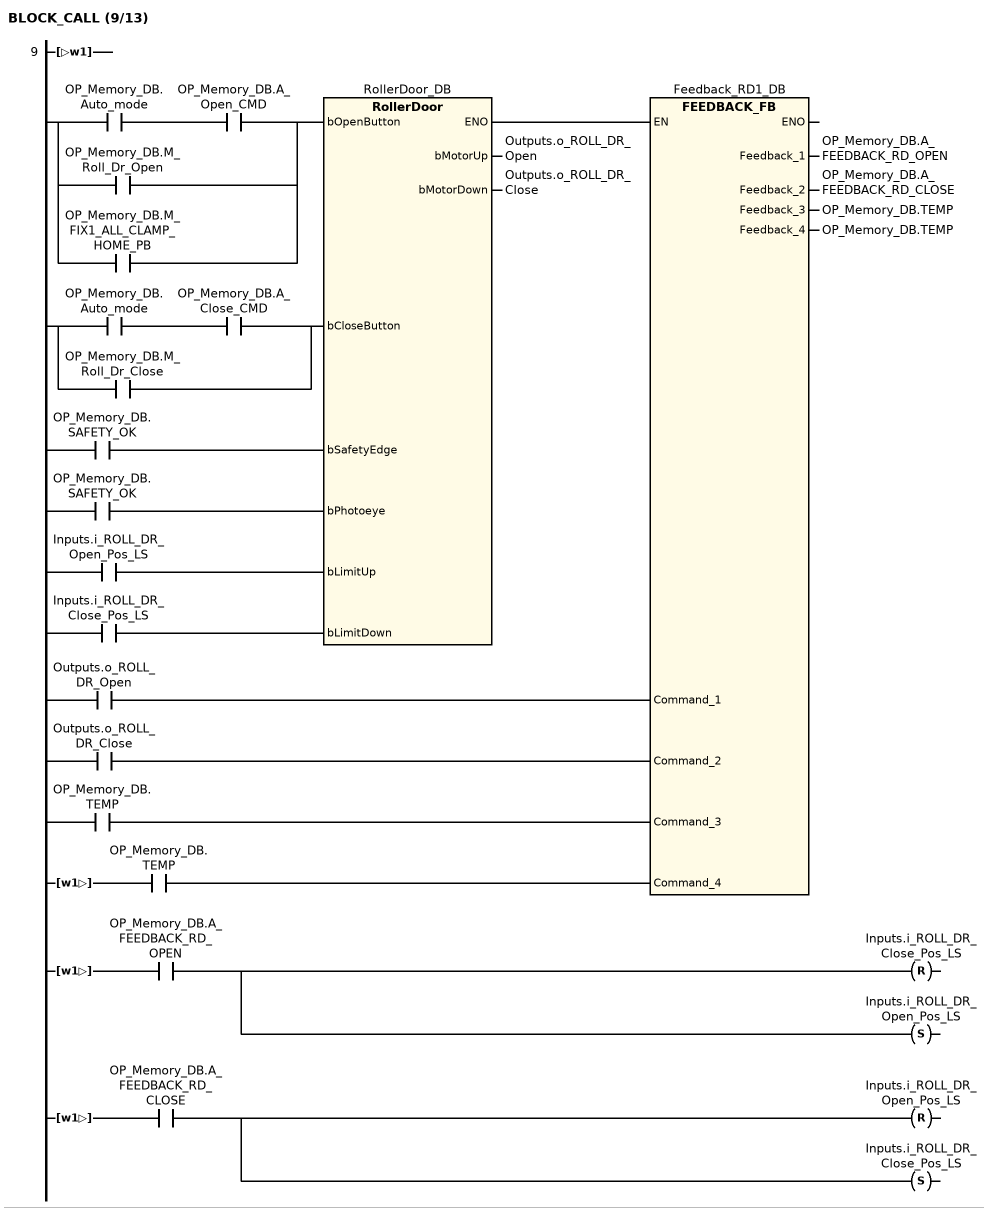
// NETWORK 9
RollerDoor_DB(
    bOpenButton := OP_Memory_DB.Auto_mode AND OP_Memory_DB.A_Open_CMD OR OP_Memory_DB.M_Roll_Dr_Open OR OP_Memory_DB.M_FIX1_ALL_CLAMP_HOME_PB,
    bCloseButton := OP_Memory_DB.Auto_mode AND OP_Memory_DB.A_Close_CMD OR OP_Memory_DB.M_Roll_Dr_Close,
    bSafetyEdge := OP_Memory_DB.SAFETY_OK,
    bPhotoeye := OP_Memory_DB.SAFETY_OK,
    bLimitUp := Inputs.i_ROLL_DR_Open_Pos_LS,
    bLimitDown := Inputs.i_ROLL_DR_Close_Pos_LS,
    bMotorUp => Outputs.o_ROLL_DR_Open,
    bMotorDown => Outputs.o_ROLL_DR_Close); // RollerDoor
Feedback_RD1_DB(
    EN := TRUE,
    Command_1 := Outputs.o_ROLL_DR_Open,
    Command_2 := Outputs.o_ROLL_DR_Close,
    Command_3 := OP_Memory_DB.TEMP,
    Command_4 := OP_Memory_DB.TEMP,
    Feedback_1 => OP_Memory_DB.A_FEEDBACK_RD_OPEN,
    Feedback_2 => OP_Memory_DB.A_FEEDBACK_RD_CLOSE,
    Feedback_3 => OP_Memory_DB.TEMP,
    Feedback_4 => OP_Memory_DB.TEMP); // FEEDBACK_FB
Inputs.i_ROLL_DR_Close_Pos_LS R= OP_Memory_DB.A_FEEDBACK_RD_OPEN;
Inputs.i_ROLL_DR_Open_Pos_LS S= OP_Memory_DB.A_FEEDBACK_RD_OPEN;
Inputs.i_ROLL_DR_Open_Pos_LS R= OP_Memory_DB.A_FEEDBACK_RD_CLOSE;
Inputs.i_ROLL_DR_Close_Pos_LS S= OP_Memory_DB.A_FEEDBACK_RD_CLOSE;

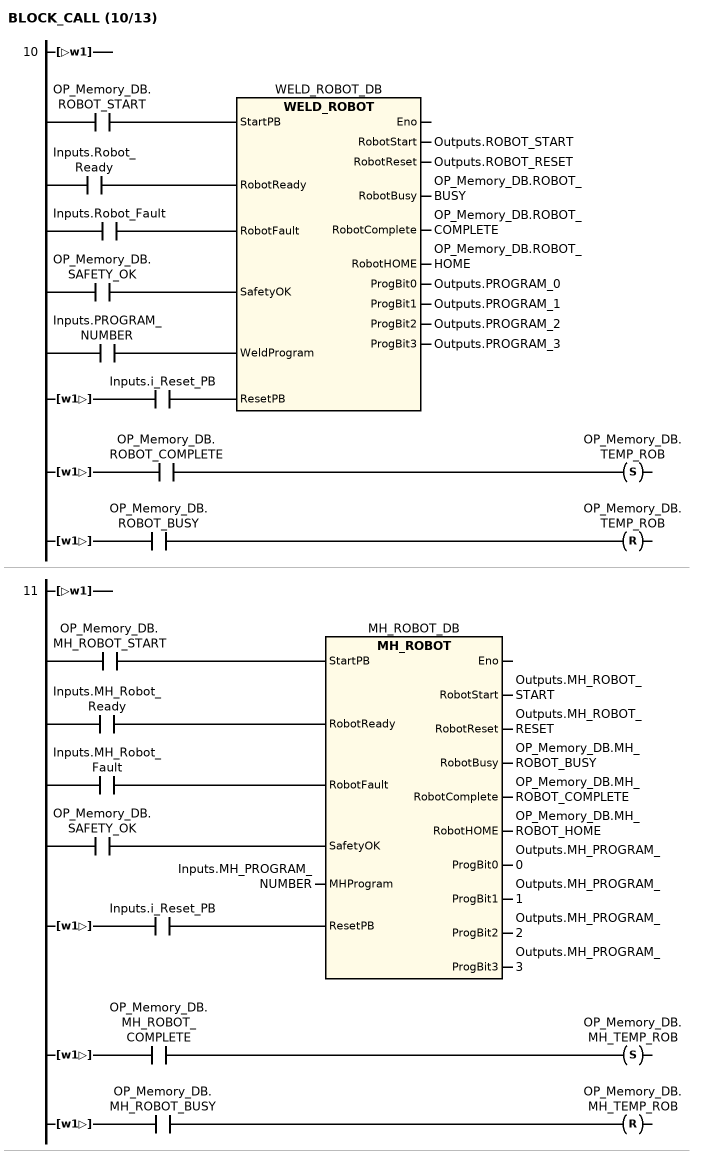
// NETWORK 10
WELD_ROBOT_DB(
    StartPB := OP_Memory_DB.ROBOT_START,
    RobotReady := Inputs.Robot_Ready,
    RobotFault := Inputs.Robot_Fault,
    SafetyOK := OP_Memory_DB.SAFETY_OK,
    WeldProgram := Inputs.PROGRAM_NUMBER,
    ResetPB := Inputs.i_Reset_PB,
    RobotStart => Outputs.ROBOT_START,
    RobotReset => Outputs.ROBOT_RESET,
    RobotBusy => OP_Memory_DB.ROBOT_BUSY,
    RobotComplete => OP_Memory_DB.ROBOT_COMPLETE,
    RobotHOME => OP_Memory_DB.ROBOT_HOME,
    ProgBit0 => Outputs.PROGRAM_0,
    ProgBit1 => Outputs.PROGRAM_1,
    ProgBit2 => Outputs.PROGRAM_2,
    ProgBit3 => Outputs.PROGRAM_3); // WELD_ROBOT
OP_Memory_DB.TEMP_ROB S= OP_Memory_DB.ROBOT_COMPLETE;
OP_Memory_DB.TEMP_ROB R= OP_Memory_DB.ROBOT_BUSY;

// NETWORK 11
MH_ROBOT_DB(
    StartPB := OP_Memory_DB.MH_ROBOT_START,
    RobotReady := Inputs.MH_Robot_Ready,
    RobotFault := Inputs.MH_Robot_Fault,
    SafetyOK := OP_Memory_DB.SAFETY_OK,
    MHProgram := Inputs.MH_PROGRAM_NUMBER,
    ResetPB := Inputs.i_Reset_PB,
    RobotStart => Outputs.MH_ROBOT_START,
    RobotReset => Outputs.MH_ROBOT_RESET,
    RobotBusy => OP_Memory_DB.MH_ROBOT_BUSY,
    RobotComplete => OP_Memory_DB.MH_ROBOT_COMPLETE,
    RobotHOME => OP_Memory_DB.MH_ROBOT_HOME,
    ProgBit0 => Outputs.MH_PROGRAM_0,
    ProgBit1 => Outputs.MH_PROGRAM_1,
    ProgBit2 => Outputs.MH_PROGRAM_2,
    ProgBit3 => Outputs.MH_PROGRAM_3); // MH_ROBOT
OP_Memory_DB.MH_TEMP_ROB S= OP_Memory_DB.MH_ROBOT_COMPLETE;
OP_Memory_DB.MH_TEMP_ROB R= OP_Memory_DB.MH_ROBOT_BUSY;

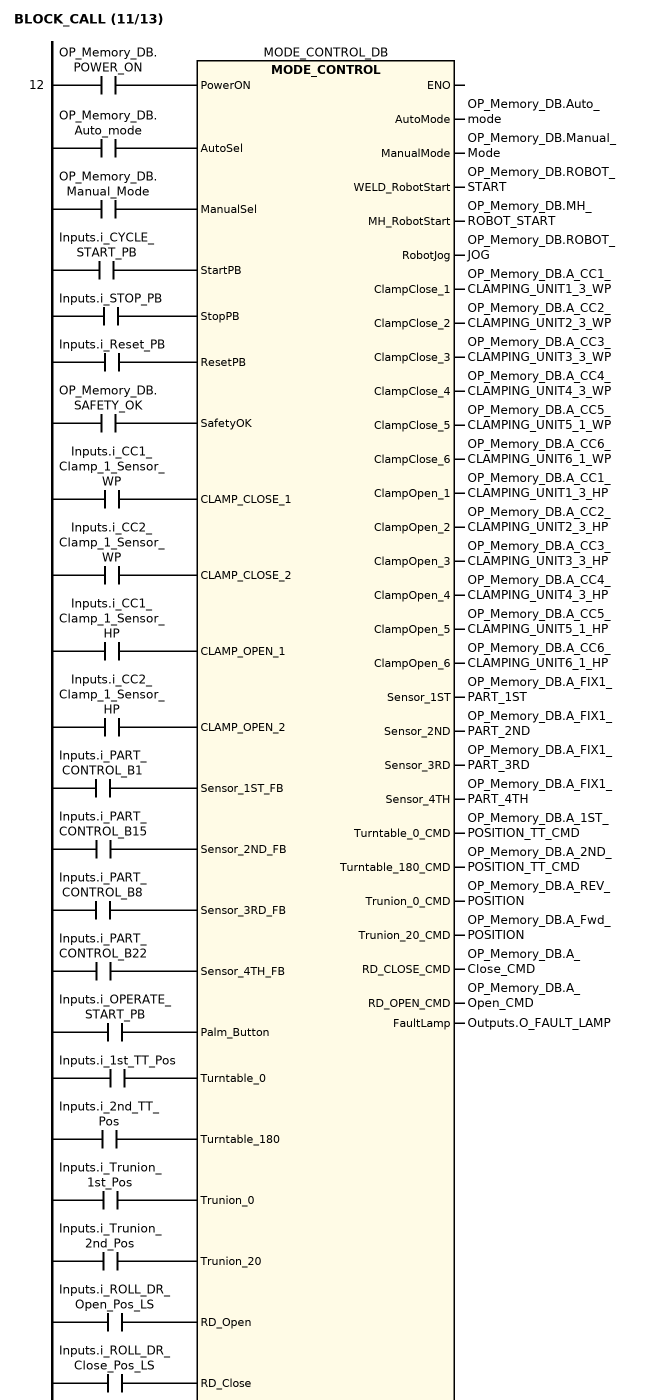
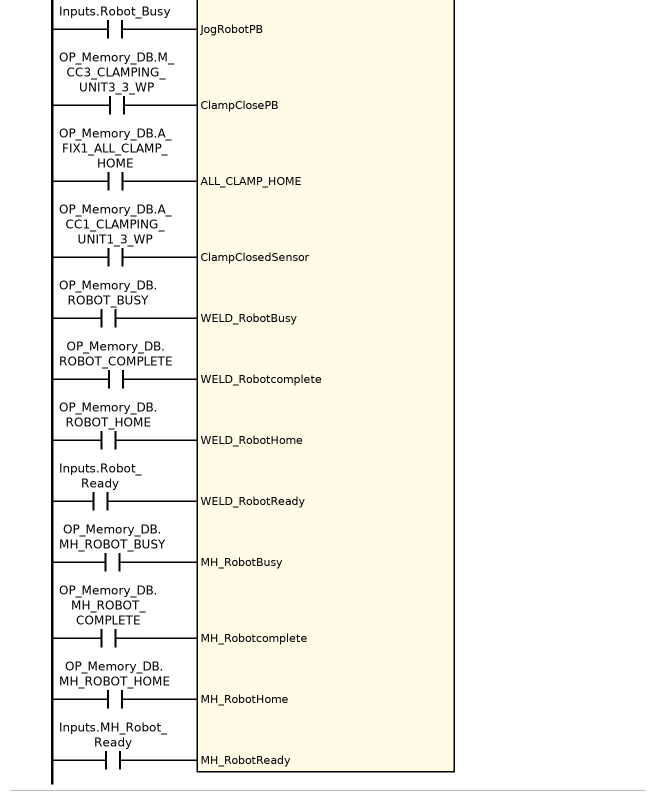
// NETWORK 12
MODE_CONTROL_DB(
    PowerON := OP_Memory_DB.POWER_ON,
    AutoSel := OP_Memory_DB.Auto_mode,
    ManualSel := OP_Memory_DB.Manual_Mode,
    StartPB := Inputs.i_CYCLE_START_PB,
    StopPB := Inputs.i_STOP_PB,
    ResetPB := Inputs.i_Reset_PB,
    SafetyOK := OP_Memory_DB.SAFETY_OK,
    CLAMP_CLOSE_1 := Inputs.i_CC1_Clamp_1_Sensor_WP,
    CLAMP_CLOSE_2 := Inputs.i_CC2_Clamp_1_Sensor_WP,
    CLAMP_OPEN_1 := Inputs.i_CC1_Clamp_1_Sensor_HP,
    CLAMP_OPEN_2 := Inputs.i_CC2_Clamp_1_Sensor_HP,
    Sensor_1ST_FB := Inputs.i_PART_CONTROL_B1,
    Sensor_2ND_FB := Inputs.i_PART_CONTROL_B15,
    Sensor_3RD_FB := Inputs.i_PART_CONTROL_B8,
    Sensor_4TH_FB := Inputs.i_PART_CONTROL_B22,
    Palm_Button := Inputs.i_OPERATE_START_PB,
    Turntable_0 := Inputs.i_1st_TT_Pos,
    Turntable_180 := Inputs.i_2nd_TT_Pos,
    Trunion_0 := Inputs.i_Trunion_1st_Pos,
    Trunion_20 := Inputs.i_Trunion_2nd_Pos,
    RD_Open := Inputs.i_ROLL_DR_Open_Pos_LS,
    RD_Close := Inputs.i_ROLL_DR_Close_Pos_LS,
    JogRobotPB := Inputs.Robot_Busy,
    ClampClosePB := OP_Memory_DB.M_CC3_CLAMPING_UNIT3_3_WP,
    ALL_CLAMP_HOME := OP_Memory_DB.A_FIX1_ALL_CLAMP_HOME,
    ClampClosedSensor := OP_Memory_DB.A_CC1_CLAMPING_UNIT1_3_WP,
    WELD_RobotBusy := OP_Memory_DB.ROBOT_BUSY,
    WELD_Robotcomplete := OP_Memory_DB.ROBOT_COMPLETE,
    WELD_RobotHome := OP_Memory_DB.ROBOT_HOME,
    WELD_RobotReady := Inputs.Robot_Ready,
    MH_RobotBusy := OP_Memory_DB.MH_ROBOT_BUSY,
    MH_Robotcomplete := OP_Memory_DB.MH_ROBOT_COMPLETE,
    MH_RobotHome := OP_Memory_DB.MH_ROBOT_HOME,
    MH_RobotReady := Inputs.MH_Robot_Ready,
    AutoMode => OP_Memory_DB.Auto_mode,
    ManualMode => OP_Memory_DB.Manual_Mode,
    WELD_RobotStart => OP_Memory_DB.ROBOT_START,
    MH_RobotStart => OP_Memory_DB.MH_ROBOT_START,
    RobotJog => OP_Memory_DB.ROBOT_JOG,
    ClampClose_1 => OP_Memory_DB.A_CC1_CLAMPING_UNIT1_3_WP,
    ClampClose_2 => OP_Memory_DB.A_CC2_CLAMPING_UNIT2_3_WP,
    ClampClose_3 => OP_Memory_DB.A_CC3_CLAMPING_UNIT3_3_WP,
    ClampClose_4 => OP_Memory_DB.A_CC4_CLAMPING_UNIT4_3_WP,
    ClampClose_5 => OP_Memory_DB.A_CC5_CLAMPING_UNIT5_1_WP,
    ClampClose_6 => OP_Memory_DB.A_CC6_CLAMPING_UNIT6_1_WP,
    ClampOpen_1 => OP_Memory_DB.A_CC1_CLAMPING_UNIT1_3_HP,
    ClampOpen_2 => OP_Memory_DB.A_CC2_CLAMPING_UNIT2_3_HP,
    ClampOpen_3 => OP_Memory_DB.A_CC3_CLAMPING_UNIT3_3_HP,
    ClampOpen_4 => OP_Memory_DB.A_CC4_CLAMPING_UNIT4_3_HP,
    ClampOpen_5 => OP_Memory_DB.A_CC5_CLAMPING_UNIT5_1_HP,
    ClampOpen_6 => OP_Memory_DB.A_CC6_CLAMPING_UNIT6_1_HP,
    Sensor_1ST => OP_Memory_DB.A_FIX1_PART_1ST,
    Sensor_2ND => OP_Memory_DB.A_FIX1_PART_2ND,
    Sensor_3RD => OP_Memory_DB.A_FIX1_PART_3RD,
    Sensor_4TH => OP_Memory_DB.A_FIX1_PART_4TH,
    Turntable_0_CMD => OP_Memory_DB.A_1ST_POSITION_TT_CMD,
    Turntable_180_CMD => OP_Memory_DB.A_2ND_POSITION_TT_CMD,
    Trunion_0_CMD => OP_Memory_DB.A_REV_POSITION,
    Trunion_20_CMD => OP_Memory_DB.A_Fwd_POSITION,
    RD_CLOSE_CMD => OP_Memory_DB.A_Close_CMD,
    RD_OPEN_CMD => OP_Memory_DB.A_Open_CMD,
    FaultLamp => Outputs.O_FAULT_LAMP); // MODE_CONTROL

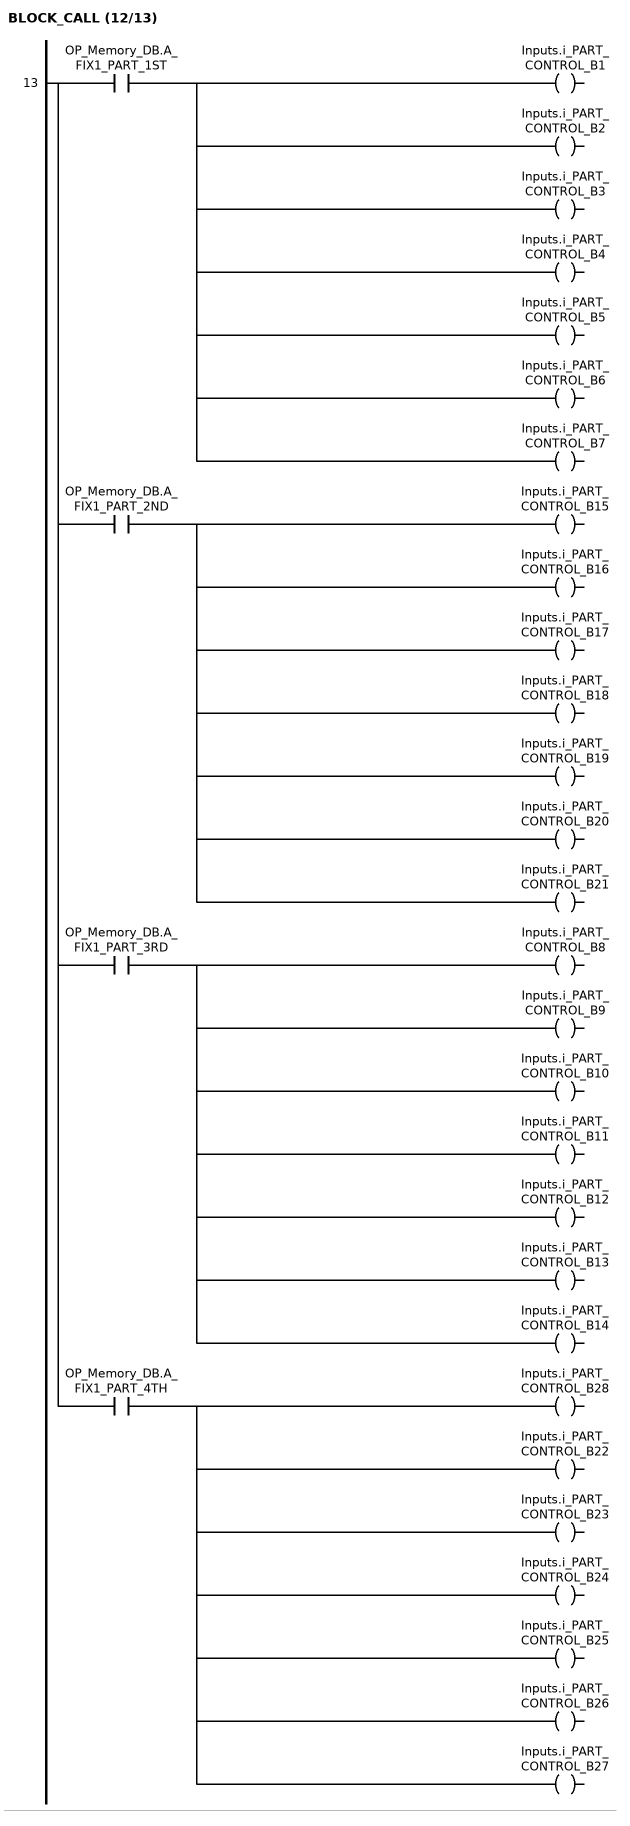
// NETWORK 13
Inputs.i_PART_CONTROL_B1 := OP_Memory_DB.A_FIX1_PART_1ST;
Inputs.i_PART_CONTROL_B2 := OP_Memory_DB.A_FIX1_PART_1ST;
Inputs.i_PART_CONTROL_B3 := OP_Memory_DB.A_FIX1_PART_1ST;
Inputs.i_PART_CONTROL_B4 := OP_Memory_DB.A_FIX1_PART_1ST;
Inputs.i_PART_CONTROL_B5 := OP_Memory_DB.A_FIX1_PART_1ST;
Inputs.i_PART_CONTROL_B6 := OP_Memory_DB.A_FIX1_PART_1ST;
Inputs.i_PART_CONTROL_B7 := OP_Memory_DB.A_FIX1_PART_1ST;
Inputs.i_PART_CONTROL_B15 := OP_Memory_DB.A_FIX1_PART_2ND;
Inputs.i_PART_CONTROL_B16 := OP_Memory_DB.A_FIX1_PART_2ND;
Inputs.i_PART_CONTROL_B17 := OP_Memory_DB.A_FIX1_PART_2ND;
Inputs.i_PART_CONTROL_B18 := OP_Memory_DB.A_FIX1_PART_2ND;
Inputs.i_PART_CONTROL_B19 := OP_Memory_DB.A_FIX1_PART_2ND;
Inputs.i_PART_CONTROL_B20 := OP_Memory_DB.A_FIX1_PART_2ND;
Inputs.i_PART_CONTROL_B21 := OP_Memory_DB.A_FIX1_PART_2ND;
Inputs.i_PART_CONTROL_B8 := OP_Memory_DB.A_FIX1_PART_3RD;
Inputs.i_PART_CONTROL_B9 := OP_Memory_DB.A_FIX1_PART_3RD;
Inputs.i_PART_CONTROL_B10 := OP_Memory_DB.A_FIX1_PART_3RD;
Inputs.i_PART_CONTROL_B11 := OP_Memory_DB.A_FIX1_PART_3RD;
Inputs.i_PART_CONTROL_B12 := OP_Memory_DB.A_FIX1_PART_3RD;
Inputs.i_PART_CONTROL_B13 := OP_Memory_DB.A_FIX1_PART_3RD;
Inputs.i_PART_CONTROL_B14 := OP_Memory_DB.A_FIX1_PART_3RD;
Inputs.i_PART_CONTROL_B28 := OP_Memory_DB.A_FIX1_PART_4TH;
Inputs.i_PART_CONTROL_B22 := OP_Memory_DB.A_FIX1_PART_4TH;
Inputs.i_PART_CONTROL_B23 := OP_Memory_DB.A_FIX1_PART_4TH;
Inputs.i_PART_CONTROL_B24 := OP_Memory_DB.A_FIX1_PART_4TH;
Inputs.i_PART_CONTROL_B25 := OP_Memory_DB.A_FIX1_PART_4TH;
Inputs.i_PART_CONTROL_B26 := OP_Memory_DB.A_FIX1_PART_4TH;
Inputs.i_PART_CONTROL_B27 := OP_Memory_DB.A_FIX1_PART_4TH;

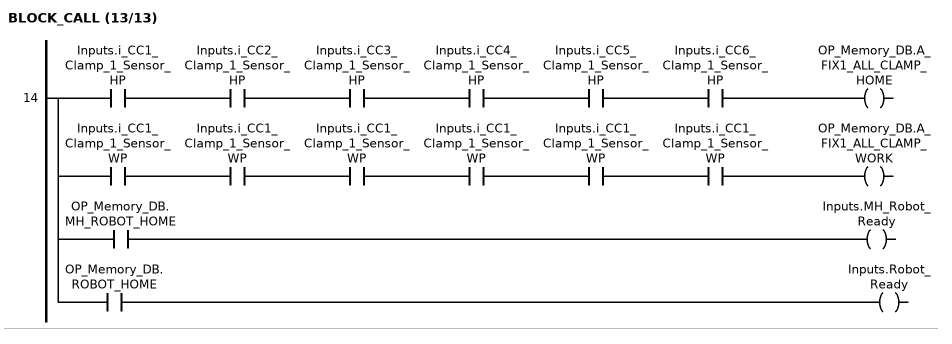
// NETWORK 14
OP_Memory_DB.A_FIX1_ALL_CLAMP_HOME := ((((Inputs.i_CC1_Clamp_1_Sensor_HP AND Inputs.i_CC2_Clamp_1_Sensor_HP) AND Inputs.i_CC3_Clamp_1_Sensor_HP) AND Inputs.i_CC4_Clamp_1_Sensor_HP) AND Inputs.i_CC5_Clamp_1_Sensor_HP) AND Inputs.i_CC6_Clamp_1_Sensor_HP;
OP_Memory_DB.A_FIX1_ALL_CLAMP_WORK := ((((Inputs.i_CC1_Clamp_1_Sensor_WP AND Inputs.i_CC1_Clamp_1_Sensor_WP) AND Inputs.i_CC1_Clamp_1_Sensor_WP) AND Inputs.i_CC1_Clamp_1_Sensor_WP) AND Inputs.i_CC1_Clamp_1_Sensor_WP) AND Inputs.i_CC1_Clamp_1_Sensor_WP;
Inputs.MH_Robot_Ready := OP_Memory_DB.MH_ROBOT_HOME;
Inputs.Robot_Ready := OP_Memory_DB.ROBOT_HOME;

END_PROGRAM

(* stored: Version 1.1.0.1, ProductVersion 3.1.4024.16
   POU BLOCK_CALL: Id {6c615bca-ca39-433d-9026-52fe92c31af4}, SpecialFunc None *)
